PROGRAM MAIN
VAR
	FCS  : BOOL := FALSE;
	FCC : BOOL := FALSE;
	FCA  : BOOL := FALSE;
	FCB  : BOOL := FALSE;
	FC1 : BOOL := FALSE;
	FC2 : BOOL := FALSE;
	START  : BOOL := FALSE;
	RESET  : BOOL := FALSE;
	BRACCIOSUP  : BOOL := FALSE;
	BRACCIOINF : BOOL := FALSE;
	DX : BOOL := FALSE;
	SX : BOOL := FALSE;
	SU : BOOL := FALSE;
	GIU : BOOL := FALSE;
	CARICATO1 : BOOL := FALSE;
	CARICATO2 : BOOL := FALSE;
	M1 : BOOL := FALSE;
	M2 : BOOL := FALSE;
	P1 : BOOL := FALSE;
	P2 : BOOL := FALSE;
	G1 : BOOL := FALSE; //GIACCA
	G2 : BOOL := FALSE; //FELPA
	S1 : BOOL := FALSE;
	S2 : BOOL := FALSE;
	ALLARME : BOOL := FALSE;
	T_ALLARME : TIME := T#30S;
END_VAR

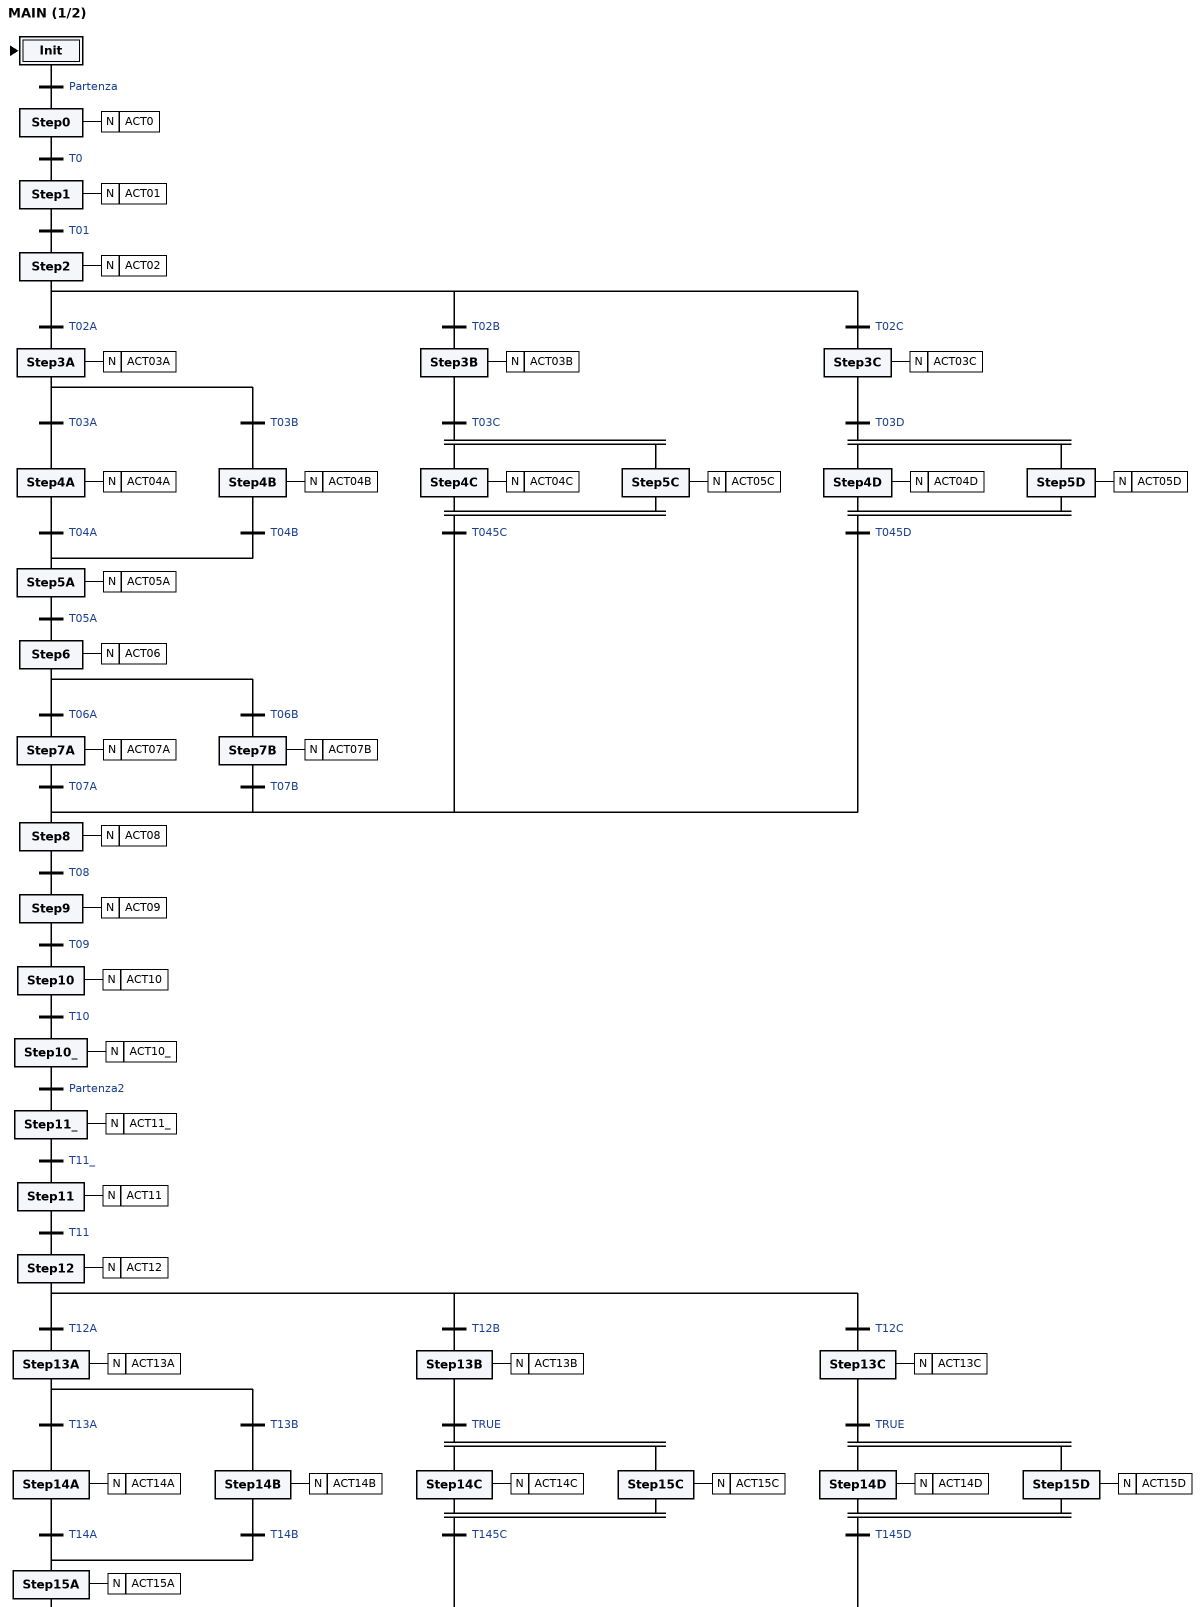
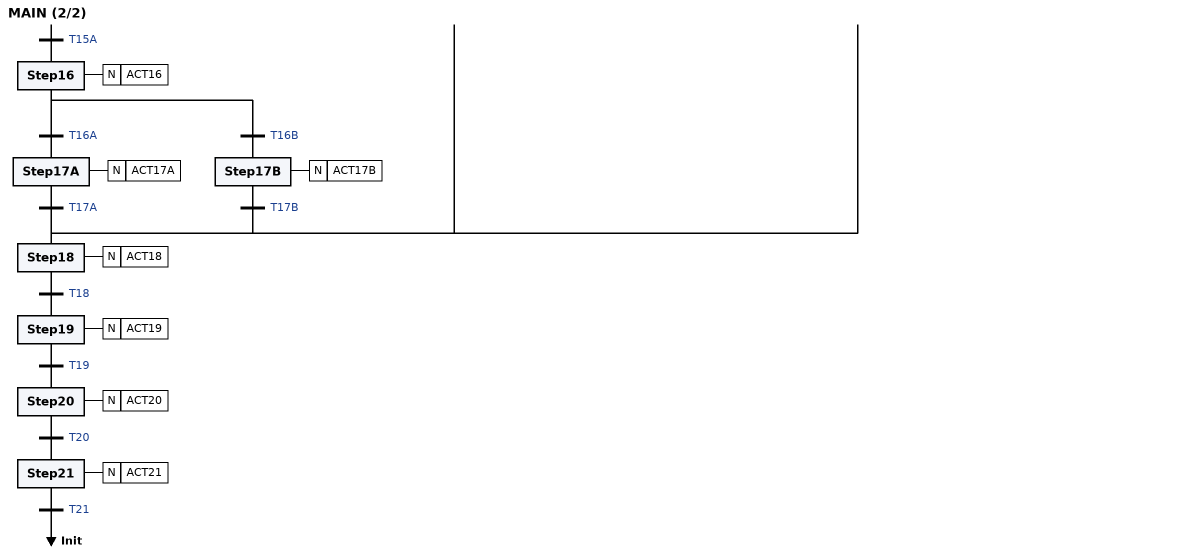
INITIAL_STEP Init:
END_STEP
TRANSITION FROM Init TO Step0
    := Partenza;
END_TRANSITION
STEP Step0:
    ACT0(N);
END_STEP
TRANSITION FROM Step0 TO Step1
    := T0;
END_TRANSITION
STEP Step1:
    ACT01(N);
END_STEP
TRANSITION FROM Step1 TO Step2
    := T01;
END_TRANSITION
STEP Step2:
    ACT02(N);
END_STEP
TRANSITION FROM Step2 TO Step3A
    := T02A;
END_TRANSITION
STEP Step3A:
    ACT03A(N);
END_STEP
TRANSITION FROM Step3A TO Step4A
    := T03A;
END_TRANSITION
STEP Step4A:
    ACT04A(N);
END_STEP
TRANSITION FROM Step4A TO Step5A
    := T04A;
END_TRANSITION
TRANSITION FROM Step3A TO Step4B
    := T03B;
END_TRANSITION
STEP Step4B:
    ACT04B(N);
END_STEP
TRANSITION FROM Step4B TO Step5A
    := T04B;
END_TRANSITION
STEP Step5A:
    ACT05A(N);
END_STEP
TRANSITION FROM Step5A TO Step6
    := T05A;
END_TRANSITION
STEP Step6:
    ACT06(N);
END_STEP
TRANSITION FROM Step6 TO Step7A
    := T06A;
END_TRANSITION
STEP Step7A:
    ACT07A(N);
END_STEP
TRANSITION FROM Step7A TO Step8
    := T07A;
END_TRANSITION
TRANSITION FROM Step6 TO Step7B
    := T06B;
END_TRANSITION
STEP Step7B:
    ACT07B(N);
END_STEP
TRANSITION FROM Step7B TO Step8
    := T07B;
END_TRANSITION
TRANSITION FROM Step2 TO Step3B
    := T02B;
END_TRANSITION
STEP Step3B:
    ACT03B(N);
END_STEP
TRANSITION FROM Step3B TO (Step4C, Step5C)
    := T03C;
END_TRANSITION
STEP Step4C:
    ACT04C(N);
END_STEP
STEP Step5C:
    ACT05C(N);
END_STEP
TRANSITION FROM (Step4C, Step5C) TO Step8
    := T045C;
END_TRANSITION
TRANSITION FROM Step2 TO Step3C
    := T02C;
END_TRANSITION
STEP Step3C:
    ACT03C(N);
END_STEP
TRANSITION FROM Step3C TO (Step4D, Step5D)
    := T03D;
END_TRANSITION
STEP Step4D:
    ACT04D(N);
END_STEP
STEP Step5D:
    ACT05D(N);
END_STEP
TRANSITION FROM (Step4D, Step5D) TO Step8
    := T045D;
END_TRANSITION
STEP Step8:
    ACT08(N);
END_STEP
TRANSITION FROM Step8 TO Step9
    := T08;
END_TRANSITION
STEP Step9:
    ACT09(N);
END_STEP
TRANSITION FROM Step9 TO Step10
    := T09;
END_TRANSITION
STEP Step10:
    ACT10(N);
END_STEP
TRANSITION FROM Step10 TO Step10_
    := T10;
END_TRANSITION
STEP Step10_:
    ACT10_(N);
END_STEP
TRANSITION FROM Step10_ TO Step11_
    := Partenza2;
END_TRANSITION
STEP Step11_:
    ACT11_(N);
END_STEP
TRANSITION FROM Step11_ TO Step11
    := T11_;
END_TRANSITION
STEP Step11:
    ACT11(N);
END_STEP
TRANSITION FROM Step11 TO Step12
    := T11;
END_TRANSITION
STEP Step12:
    ACT12(N);
END_STEP
TRANSITION FROM Step12 TO Step13A
    := T12A;
END_TRANSITION
STEP Step13A:
    ACT13A(N);
END_STEP
TRANSITION FROM Step13A TO Step14A
    := T13A;
END_TRANSITION
STEP Step14A:
    ACT14A(N);
END_STEP
TRANSITION FROM Step14A TO Step15A
    := T14A;
END_TRANSITION
TRANSITION FROM Step13A TO Step14B
    := T13B;
END_TRANSITION
STEP Step14B:
    ACT14B(N);
END_STEP
TRANSITION FROM Step14B TO Step15A
    := T14B;
END_TRANSITION
STEP Step15A:
    ACT15A(N);
END_STEP
TRANSITION FROM Step15A TO Step16
    := T15A;
END_TRANSITION
STEP Step16:
    ACT16(N);
END_STEP
TRANSITION FROM Step16 TO Step17A
    := T16A;
END_TRANSITION
STEP Step17A:
    ACT17A(N);
END_STEP
TRANSITION FROM Step17A TO Step18
    := T17A;
END_TRANSITION
TRANSITION FROM Step16 TO Step17B
    := T16B;
END_TRANSITION
STEP Step17B:
    ACT17B(N);
END_STEP
TRANSITION FROM Step17B TO Step18
    := T17B;
END_TRANSITION
TRANSITION FROM Step12 TO Step13B
    := T12B;
END_TRANSITION
STEP Step13B:
    ACT13B(N);
END_STEP
TRANSITION FROM Step13B TO (Step14C, Step15C)
    := TRUE;
END_TRANSITION
STEP Step14C:
    ACT14C(N);
END_STEP
STEP Step15C:
    ACT15C(N);
END_STEP
TRANSITION FROM (Step14C, Step15C) TO Step18
    := T145C;
END_TRANSITION
TRANSITION FROM Step12 TO Step13C
    := T12C;
END_TRANSITION
STEP Step13C:
    ACT13C(N);
END_STEP
TRANSITION FROM Step13C TO (Step14D, Step15D)
    := TRUE;
END_TRANSITION
STEP Step14D:
    ACT14D(N);
END_STEP
STEP Step15D:
    ACT15D(N);
END_STEP
TRANSITION FROM (Step14D, Step15D) TO Step18
    := T145D;
END_TRANSITION
STEP Step18:
    ACT18(N);
END_STEP
TRANSITION FROM Step18 TO Step19
    := T18;
END_TRANSITION
STEP Step19:
    ACT19(N);
END_STEP
TRANSITION FROM Step19 TO Step20
    := T19;
END_TRANSITION
STEP Step20:
    ACT20(N);
END_STEP
TRANSITION FROM Step20 TO Step21
    := T20;
END_TRANSITION
STEP Step21:
    ACT21(N);
END_STEP
TRANSITION FROM Step21 TO Init
    := T21;
END_TRANSITION
// branch label B01
// branch label B02
// branch label B03
// branch label B04

ACTION ACT0:
DX := TRUE;
END_ACTION

ACTION ACT01:
DX := FALSE;
SU := TRUE;
END_ACTION

ACTION ACT02:
SU := FALSE;
DX := TRUE;
END_ACTION

ACTION ACT03A:
DX := FALSE;
END_ACTION

ACTION ACT03B:
DX := FALSE;
END_ACTION

ACTION ACT03C:
DX := FALSE;
END_ACTION

ACTION ACT04A:
BRACCIOSUP := TRUE;
END_ACTION

ACTION ACT04B:
BRACCIOINF := TRUE;
END_ACTION

ACTION ACT04C:
BRACCIOSUP := TRUE;
END_ACTION

ACTION ACT04D:
BRACCIOSUP := TRUE;
END_ACTION

ACTION ACT05A:
DX := TRUE;
BRACCIOSUP := FALSE;
BRACCIOINF := FALSE;
END_ACTION

ACTION ACT05C:
BRACCIOINF := TRUE;
END_ACTION

ACTION ACT05D:
BRACCIOINF := TRUE;
END_ACTION

ACTION ACT06:
DX := FALSE;
END_ACTION

ACTION ACT07A:
BRACCIOSUP := TRUE;
END_ACTION

ACTION ACT07B:
BRACCIOINF := TRUE;
END_ACTION

ACTION ACT08:
SX := TRUE;
BRACCIOSUP := FALSE;
BRACCIOINF := FALSE;
END_ACTION

ACTION ACT09:
SX := FALSE;
GIU := TRUE;
END_ACTION

ACTION ACT10:
GIU := FALSE;
SX := TRUE;
END_ACTION

ACTION ACT10_:
SX := FALSE;
END_ACTION

ACTION ACT11:
GIU := TRUE;
DX := FALSE;
END_ACTION

ACTION ACT11_:
DX := TRUE;
END_ACTION

ACTION ACT12:
GIU := FALSE;
DX := TRUE;
END_ACTION

ACTION ACT13A:
DX := FALSE;
END_ACTION

ACTION ACT13B:
DX := FALSE;
END_ACTION

ACTION ACT13C:
DX := FALSE;
END_ACTION

ACTION ACT14A:
BRACCIOSUP := TRUE;
END_ACTION

ACTION ACT14B:
BRACCIOINF := TRUE;
END_ACTION

ACTION ACT14C:
BRACCIOSUP := TRUE;
END_ACTION

ACTION ACT14D:
BRACCIOSUP := TRUE;
END_ACTION

ACTION ACT15A:
DX := TRUE;
BRACCIOSUP := FALSE;
BRACCIOINF := FALSE;
END_ACTION

ACTION ACT15C:
BRACCIOINF := TRUE;
END_ACTION

ACTION ACT15D:
BRACCIOINF := TRUE;
END_ACTION

ACTION ACT16:
DX := FALSE;
END_ACTION

ACTION ACT17A:
BRACCIOSUP := TRUE;
END_ACTION

ACTION ACT17B:
BRACCIOINF := TRUE;
END_ACTION

ACTION ACT18:
SX := TRUE;
BRACCIOSUP := FALSE;
BRACCIOINF := FALSE;
END_ACTION

ACTION ACT19:
SX := FALSE;
SU := TRUE;
END_ACTION

ACTION ACT20:
SX := TRUE;
SU := FALSE;
END_ACTION

ACTION ACT21:
SX := FALSE;
END_ACTION

TRANSITION Partenza:
START AND ((M1 XOR M2) AND (P1 XOR P2)) ;
END_TRANSITION

TRANSITION Partenza2:
(NOT CARICATO1) AND (NOT CARICATO2) AND ((G1 XOR G2) AND (S1 XOR S2));
END_TRANSITION

TRANSITION T0:
FCC;
END_TRANSITION

TRANSITION T01:
FCA;
END_TRANSITION

TRANSITION T02A:
(FC1 AND (M1 XOR P1));
END_TRANSITION

TRANSITION T02B:
FC1 AND (M1 AND P1);
END_TRANSITION

TRANSITION T02C:
FC2 AND M2 AND P2;
END_TRANSITION

TRANSITION T03A:
M1;
END_TRANSITION

TRANSITION T03B:
P1;
END_TRANSITION

TRANSITION T03C:
TRUE;
END_TRANSITION

TRANSITION T03D:
TRUE;
END_TRANSITION

TRANSITION T045C:
CARICATO1 AND CARICATO2;
END_TRANSITION

TRANSITION T045D:
CARICATO1 AND CARICATO2;
END_TRANSITION

TRANSITION T04A:
CARICATO1;
END_TRANSITION

TRANSITION T04B:
CARICATO2;
END_TRANSITION

TRANSITION T05A:
FC2 AND (M2 OR P2);
END_TRANSITION

TRANSITION T06A:
M2;
END_TRANSITION

TRANSITION T06B:
P2;
END_TRANSITION

TRANSITION T07A:
CARICATO1;
END_TRANSITION

TRANSITION T07B:
CARICATO2;
END_TRANSITION

TRANSITION T08:
FCA;
END_TRANSITION

TRANSITION T09:
FCC;
END_TRANSITION

TRANSITION T10:
FCS;
END_TRANSITION

TRANSITION T11:
FCB;
END_TRANSITION

TRANSITION T11_:
FCC;
END_TRANSITION

TRANSITION T12A:
FC1 AND (G1 XOR S1)
END_TRANSITION

TRANSITION T12B:
FC1 AND (G1 AND S1);
END_TRANSITION

TRANSITION T12C:
FC2 AND (G2 AND S2);
END_TRANSITION

TRANSITION T13A:
G1;
END_TRANSITION

TRANSITION T13B:
S1;
END_TRANSITION

TRANSITION T145C:
CARICATO1 AND CARICATO2;
END_TRANSITION

TRANSITION T145D:
CARICATO1 AND CARICATO2;
END_TRANSITION

TRANSITION T14A:
CARICATO1;
END_TRANSITION

TRANSITION T14B:
CARICATO2;
END_TRANSITION

TRANSITION T15A:
FC2 AND (G2 XOR S2);
END_TRANSITION

TRANSITION T16A:
G2;
END_TRANSITION

TRANSITION T16B:
S2;
END_TRANSITION

TRANSITION T17A:
CARICATO1;
END_TRANSITION

TRANSITION T17B:
CARICATO2;
END_TRANSITION

TRANSITION T18:
FCB;
END_TRANSITION

TRANSITION T19:
FCC;
END_TRANSITION

TRANSITION T20:
FCS;
END_TRANSITION

TRANSITION T21:
(NOT CARICATO1) AND (NOT CARICATO2);
END_TRANSITION

END_PROGRAM

(* stored: Version 1.1.0.1, ProductVersion 3.1.4024.10
   POU MAIN: Id {dc69dfa5-2f70-4b81-8e9e-a1adcb4fd56b}, SpecialFunc None
   Action ACT0: Id {7a8402d7-6e48-4097-9397-eca5f0b3c91a}
   Action ACT01: Id {921473b9-b143-4363-91b5-cbc3e8a927b3}
   Action ACT02: Id {195b89ef-03a5-4882-9b02-d20c59086bec}
   Action ACT03A: Id {2c4ff417-bfbc-41b1-bb87-d7eccf983c7a}
   Action ACT03B: Id {5d8f5681-992e-4358-a766-b2859eb4eb5b}
   Action ACT03C: Id {8cc5090f-e556-4b2e-83ff-a2f3fc4bc559}
   Action ACT04A: Id {530bd9c4-f9f4-4ba1-a6ef-ff9b2324773f}
   Action ACT04B: Id {2bc76db7-7145-4b54-97d6-a2e2b6c5aca2}
   Action ACT04C: Id {5295ecb7-3f69-4aca-a78d-42db20fc701f}
   Action ACT04D: Id {b0dd1c12-905c-4566-a664-c8c6d6626ca4}
   Action ACT05A: Id {9bf992e4-584f-482e-b9e8-c2ba9988c4c9}
   Action ACT05C: Id {5bf033b5-2f6c-406f-8933-bede19fc094a}
   Action ACT05D: Id {19225d0b-ce91-4e63-bc11-40b03032aa1d}
   Action ACT06: Id {ecbac40c-b4d2-4b38-9806-c54d82d4c897}
   Action ACT07A: Id {6f5eeac2-cd67-4b25-a5c6-0b224396f644}
   Action ACT07B: Id {c669dd07-dd03-4cc3-a0a0-43cedf4cb2ba}
   Action ACT08: Id {3a489772-34e1-4ce5-b46d-a00460a29a02}
   Action ACT09: Id {0bc5f5ac-5a31-45e4-94cd-a540681b9060}
   Action ACT10: Id {befb620c-2746-40a1-95bf-d5aeec8383d9}
   Action ACT10_: Id {654bf4e3-d03b-4914-9b9e-37948e5be79b}
   Action ACT11: Id {abe7f62f-e413-41a9-b34b-19c8f944249d}
   Action ACT11_: Id {fa669ee9-790e-484c-9580-b292c267c5f4}
   Action ACT12: Id {105c6e03-63ea-4ea8-9fdf-ece3abe97d8b}
   Action ACT13A: Id {f6eab527-cab8-4b53-9d3c-b773fc5d307a}
   Action ACT13B: Id {370280cf-5231-4025-9ae4-cb5e7d091521}
   Action ACT13C: Id {9be5d52a-7dea-4e19-8765-bdf3f082fe4c}
   Action ACT14A: Id {8419b164-8d8a-4cf1-84a8-0442ca2fef35}
   Action ACT14B: Id {8322037f-8166-4c76-afd7-c3f8d254b466}
   Action ACT14C: Id {5c37776b-5a2f-4f7e-9fe9-e781bf6c83e9}
   Action ACT14D: Id {196638e7-fd49-47c5-b743-7bd177607983}
   Action ACT15A: Id {8ec2c7d1-3c93-4c3a-8570-60c0c04eae67}
   Action ACT15C: Id {e262757c-09a5-4264-9595-89ef230b3bdd}
   Action ACT15D: Id {4b17b8f9-c95a-4185-8886-63269f7d8b4c}
   Action ACT16: Id {73d39081-91b0-476d-91d1-0e487ab2705d}
   Action ACT17A: Id {77b357c9-d7db-48c4-9400-d7a6da4afe13}
   Action ACT17B: Id {bb7850c3-cb82-4d5a-ad9e-c51bfff5e691}
   Action ACT18: Id {16b3e884-f6bc-41de-8132-023eb3e717ed}
   Action ACT19: Id {ab458ded-dc91-43b7-bd7d-2cddac1ca45e}
   Action ACT20: Id {5760e5a5-53ff-446d-97d6-dd5b49a438fc}
   Action ACT21: Id {0e1f9a71-2734-47f0-8300-e906add0cf26}
   Transition Partenza: Id {a4e2dcc4-e16c-40da-98d8-3cf76ee3b8ca}
   Transition Partenza2: Id {dee84d9c-b9bd-47f9-81df-ee99ba64c3af}
   Transition T0: Id {78fced0f-a212-4af7-a303-ff39d6531b4c}
   Transition T01: Id {9f44e70e-18bc-4364-9b3e-7208a03ce5a8}
   Transition T02A: Id {fb04c189-42de-41fe-b0eb-6ffe2bf85fa3}
   Transition T02B: Id {db97f07a-9130-4c25-953c-2a4d8e93de65}
   Transition T02C: Id {572d3a5a-b0a8-4ebd-a4e3-2a9ca57d84de}
   Transition T03A: Id {91884da3-0490-4624-8e56-f2f20ce5d2a8}
   Transition T03B: Id {5726b3e4-b023-4d78-9eff-6a07d54c0dd6}
   Transition T03C: Id {12d68024-9e2a-428e-a491-fddaa5ae48ee}
   Transition T03D: Id {6a06532c-c1e9-4cae-b365-81339674ff4b}
   Transition T045C: Id {555b5be8-24de-445d-bc20-b814b68e69a0}
   Transition T045D: Id {389685f5-44ac-4436-be54-44d6edab3877}
   Transition T04A: Id {84e9b1b7-097f-44d0-ae68-91c56bcfbba0}
   Transition T04B: Id {40d6b781-17f7-44ec-b80b-9060b0b56e67}
   Transition T05A: Id {a9d907c7-b688-4cd3-bf3c-88ca3134415e}
   Transition T06A: Id {e90fd188-9850-4f59-ad28-3b08c6e754d9}
   Transition T06B: Id {c8eef533-9f03-4a1e-908f-38dee8b96432}
   Transition T07A: Id {5d653ba1-1e56-46fb-bfb7-b9e525af605d}
   Transition T07B: Id {75314863-2fe6-460c-b24a-000152c771d3}
   Transition T08: Id {21829675-e53f-4791-888d-37de05240f08}
   Transition T09: Id {fcd16775-6eaa-4895-9f5d-19abe85bf523}
   Transition T10: Id {22f9778c-6e8d-4a0c-ac84-44e835ad9027}
   Transition T11: Id {6c135fda-821c-4544-9fde-95add7054f41}
   Transition T11_: Id {e071af9c-f0e5-4ef5-a064-d20bf584eab3}
   Transition T12A: Id {20505384-851c-45c9-81f5-17bfdae968b7}
   Transition T12B: Id {4d65f44a-bb7c-473b-8a4a-0d2264e56ff9}
   Transition T12C: Id {1816b8b5-86f0-4308-bf9c-fc3357ca0c0d}
   Transition T13A: Id {984e7a77-76c9-49d1-b641-17d6fdf4016b}
   Transition T13B: Id {16a116a6-8fc9-4d53-8c6f-a80f00d68c80}
   Transition T145C: Id {e1ad5ea2-0909-4a97-b024-8186e28693c5}
   Transition T145D: Id {fdb7c401-db16-45c1-97f6-ee34c19e243b}
   Transition T14A: Id {0268c4c4-d8cb-4e74-8670-292f58615684}
   Transition T14B: Id {20f679d9-b126-468f-999b-1dff7bff798f}
   Transition T15A: Id {c5a90dde-039a-4997-874e-2cd8af58d16b}
   Transition T16A: Id {3049c26e-2a9d-4359-a6e3-ea7162da4a57}
   Transition T16B: Id {2c5e51be-9152-47be-995f-81d3ef1835de}
   Transition T17A: Id {1840291a-16d5-4471-98e6-f20a7153456a}
   Transition T17B: Id {f6a05721-8111-41fd-be8d-48131a7aadda}
   Transition T18: Id {463d3265-0dab-4e44-b044-631cb69cba9a}
   Transition T19: Id {6a847a5e-0bf9-40fa-8c25-ab00dd6444f8}
   Transition T20: Id {6f791346-e0a6-420f-b785-e45f382c21d2}
   Transition T21: Id {d7966c82-ea25-414d-8ac3-0e0f1bece6be} *)
